Fanuc KAREL source: kx00006.KL

-- PROVISIONAL review KL for V770-1; original PC SHA256 367bd63e80f20ca6e29484b9d5cfc15fadea29a7b9a1c7bc2cec3c42579aefb1
-- Incomplete behavior may be omitted. Consult companion uncertainty JSON. Do not deploy.
PROGRAM KX00006
%NOLOCKGROUP
VAR
  I : INTEGER
  J : INTEGER
  B : BOOLEAN
  F : FILE
  S : STRING[80]
-- UNRESOLVED_DECL P type=000102
BEGIN
  -- UNRESOLVED_PC offsets 5-13; opcodes 9D,2E,0F
  -- UNRESOLVED_PC offsets 18-22; opcodes 7F
END KX00006
